(* CODESYS project Soru_5.project
   Title: Adsız
   Version: 0.0.0.0
   Author: Enes

Project tree, tasks and I/O mapping:
  MyController : TM241C24T/U, Schneider Electric, order no. TM241C24T/U, version 4.0.6.18
    application Application
      task MAST (cyclic, interval 20 ms, priority 15, watchdog 100 ms x 1) calls POU
      global variables GVL
      program POU [LD]
    DI : Digital Inputs, Schneider Electric, version 4.0.6.18
        input  iwDI_IW0 : WORD  // IW0
        input  ibDI_IB1 : BYTE  // IB1
    DQ : Digital Outputs, Schneider Electric, version 4.0.6.18
        output qwDQ_QW0 : WORD  // QW0
        output qbDQ_QB1 : BYTE  // QB1
    Counters : Counters, Schneider Electric, version 4.0.6.18
    Pulse_Generators : Pulse Generators, Schneider Electric, version 4.0.6.18
    Cartridge_1 : Cartridge, Schneider Electric, version 4.0.6.18
    IO_Bus : IO bus - TM3, Schneider Electric, version 4.0.6.18
    COM_Bus : COM bus, Schneider Electric, version 4.0.6.18
    Serial_Line_1 : Serial line, Schneider Electric, version 4.0.6.18
      SoMachine_Network_Manager : SoMachine-Network Manager, Schneider Electric, version 4.0.0.2
    Serial_Line_2 : Serial line, Schneider Electric, version 4.0.6.18
      Modbus_Manager : Modbus Manager, Schneider Electric, version 4.0.0.2
*)

// MyController/Application/GVL
VAR_GLOBAL
END_VAR

// MyController/Application/POU
PROGRAM POU
VAR
	Start: BOOL;
	Stop: BOOL;
	M0: BOOL;
	Motor_2: BOOL;
	Motor_1: BOOL;
	Motor_3: BOOL;
	Timer1: TON;
	Timer2: TON;
	Timer3: TON;
	Timer4: TON;
END_VAR
VAR // added by the converter: edge detectors and wires of the graphical bodies
    _w1 : BOOL;
END_VAR

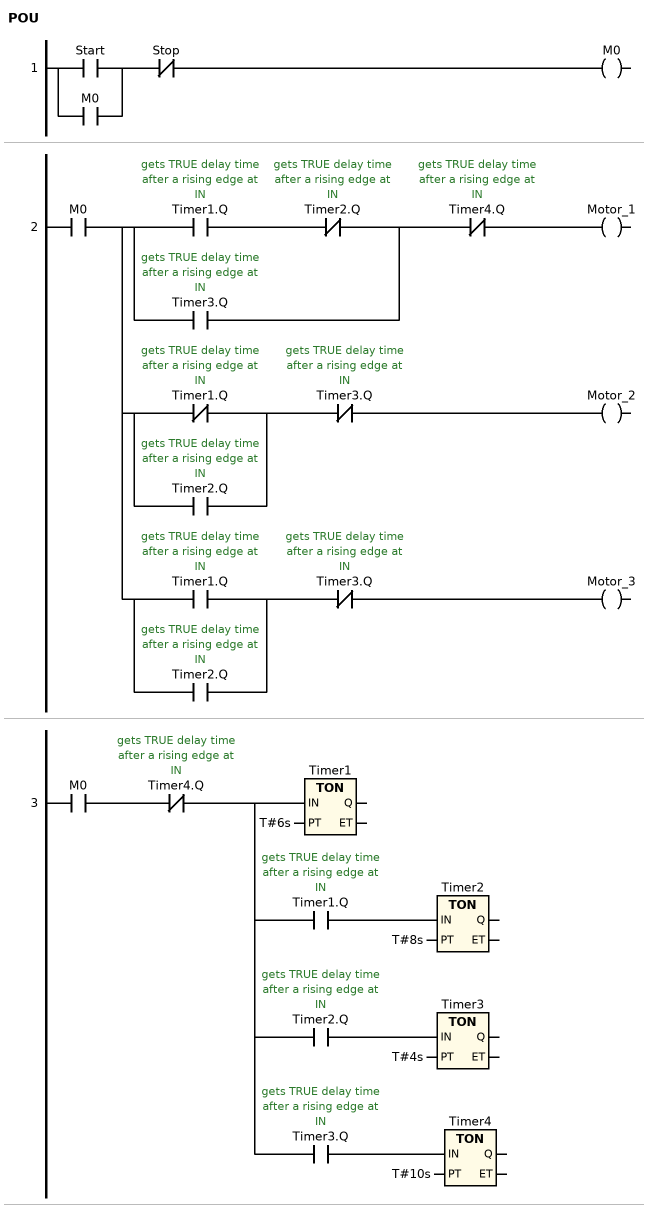
// NETWORK 1
M0 := (Start OR M0) AND NOT Stop;

// NETWORK 2
//   Timer1.Q: gets TRUE delay time after a rising edge at IN
//   Timer2.Q: gets TRUE delay time after a rising edge at IN
//   Timer3.Q: gets TRUE delay time after a rising edge at IN
//   Timer4.Q: gets TRUE delay time after a rising edge at IN
Motor_1 := M0 AND (Timer1.Q AND NOT Timer2.Q OR Timer3.Q) AND NOT Timer4.Q;
Motor_2 := M0 AND (NOT Timer1.Q OR Timer2.Q) AND NOT Timer3.Q;
Motor_3 := M0 AND (Timer1.Q OR Timer2.Q) AND NOT Timer3.Q;

// NETWORK 3
//   Timer4.Q: gets TRUE delay time after a rising edge at IN
//   Timer1.Q: gets TRUE delay time after a rising edge at IN
//   Timer2.Q: gets TRUE delay time after a rising edge at IN
//   Timer3.Q: gets TRUE delay time after a rising edge at IN
_w1 := M0 AND NOT Timer4.Q;
Timer1(IN := _w1, PT := T#6s); // TON
Timer2(IN := _w1 AND Timer1.Q, PT := T#8s); // TON
Timer3(IN := _w1 AND Timer2.Q, PT := T#4s); // TON
Timer4(IN := _w1 AND Timer3.Q, PT := T#10s); // TON

END_PROGRAM
